// TIA Portal project "ASANSÖR_BANT" (V17)
// Vorlageprojekt für das Buch mit Zielsystem S7-1200

(* hardware
DEVICE "S7-1200-Station_1"  S7-1200 Station
   slot 0: "Baugruppenträger_0"  Rack  V1.0
   slot 1: "PLC_1"  CPU 1214C DC/DC/Rly  6ES7 214-1HG40-0XB0  V4.5
*)

// ===== PLC "PLC_1"  CPU 1214C DC/DC/Rly =====

VAR_GLOBAL   // PLC tag table "Standard-Variablentabelle"
   "START" AT %E0.0 : Bool;
   "STOP" AT %E0.1 : Bool;
   "SENSÖR 1" AT %I0.2 : Bool;
   "SENSÖR 2" AT %I0.3 : Bool;
   "PLAT.LİM.SENSÖR" AT %I0.5 : Bool;
   "ASAN.LİM.SENSÖR" AT %I0.6 : Bool;
   "KONVEYÖR 1" AT %Q0.0 : Bool;
   "KONVEYÖR 2" AT %Q0.1 : Bool;
   "PLAT.İLERİ.HAR." AT %Q0.2 : Bool;
   "PLAT.DÖNDÜR" AT %Q0.3 : Bool;
   "ASAN.İLERİ" AT %Q0.4 : Bool;
   "ASAN.YUKARI" AT %Q0.5 : Bool;
   "SENSÖR 3" AT %I0.4 : Bool;
   "PLAT.DÖNÜŞ.SENSÖR" AT %I0.7 : Bool;
END_VAR

// folder: System blocks/Program resources

DATA_BLOCK "TİMER 1"   // DB1
{ S7_Optimized_Access := 'TRUE' }
AUTHOR : Simatic
FAMILY : IEC
NAME : IEC_TMR
VERSION : 1.0
// stored: InstanceOfName IEC_TIMER
"IEC_TIMER"
BEGIN
END_DATA_BLOCK

// folder: (top level)

FUNCTION "MHJ-PLC-Lab-Function-S71200" : Void   // FC9000, SCL
{ S7_Optimized_Access := 'TRUE' }
VERSION : 0.1
   VAR_TEMP
      rdTimeReturn : Int;
      outputTime : DTL;
      SyncVal : Byte;
      forVal : Int;
      forVal_2 : Int;
      Value : Byte;
   END_VAR
   VAR CONSTANT
      CompVal : Byte := 16#34;
      Value_01 : Byte := 16#11;
      Value_01_DW : DWord := 16#A165_D992;
      Value_02_DW : DWord := 16#58BE_4401;
   END_VAR
BEGIN

   #Value:=PEEK(area := 16#82,
        dbNumber := 0,
        byteOffset := 511);
   #Value := #Value + 1;

   POKE(area := 16#82,
        dbNumber := 0,
        byteOffset := 511,
        value := #Value);

   POKE(area:=16#81,
        dbNumber:=0,
        byteOffset:=1016,
        value:=#Value_01_DW);
   POKE(area := 16#81,
        dbNumber := 0,
        byteOffset := 1020,
        value := #Value_02_DW);

   POKE(area := 16#81,
        dbNumber := 0,
        byteOffset := 511,
        value := B#16#00);

   FOR #forVal := 0 TO 120 DO
       FOR #forVal_2:=0 TO 10 DO
           #rdTimeReturn:=RD_SYS_T(#outputTime);
           #rdTimeReturn := WR_SYS_T(#outputTime);
           #rdTimeReturn := RD_SYS_T(#outputTime);
           #rdTimeReturn := WR_SYS_T(#outputTime);
       END_FOR;
       #SyncVal:= PEEK(area := 16#81,
                      dbNumber := 0,
                      byteOffset := 511);
       IF #SyncVal = #CompVal THEN
          GOTO M_1;
       END_IF;
   END_FOR;
   RETURN;

   M_1:
   POKE(area := 16#81,
        dbNumber := 0,
        byteOffset := 511,
        value := B#16#0);
END_FUNCTION

ORGANIZATION_BLOCK "Main"   // OB1, LAD, ProgramCycle
TITLE = "Main Program Sweep (Cycle)"
{ S7_Optimized_Access := 'TRUE' }
VERSION : 0.1
   VAR_INPUT
      Initial_Call : Bool;   // Initial call of this OB
      Remanence : Bool;   // =True, if remanent data are available
   END_VAR
BEGIN

REGION Network 1: Konnektierungsbaustein für PLC-Lab
   // Im Netzwerk 1 wird der Konnektierungsbaustein für PLC-Lab aufgerufen.
   // Dieser Aufruf darf nicht entfernt werden!
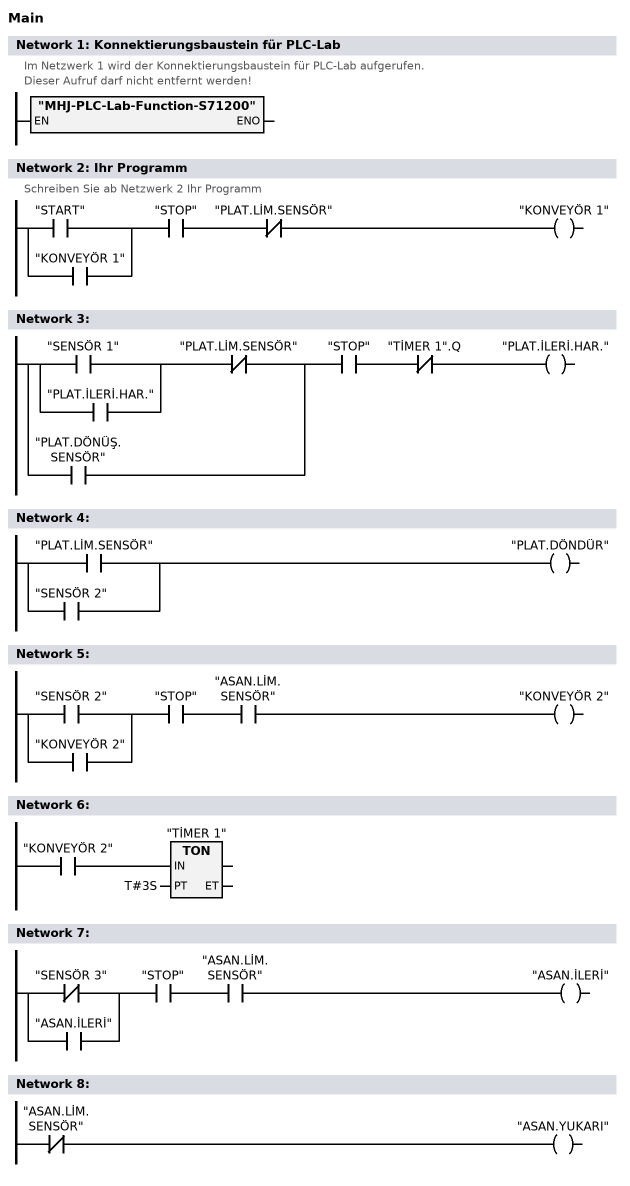
   RUNG wire#powerrail
      "MHJ-PLC-Lab-Function-S71200"()
   END_RUNG
   // the same network as SCL:
   "MHJ-PLC-Lab-Function-S71200"();
END_REGION

REGION Network 2: Ihr Programm
   // Schreiben Sie ab Netzwerk 2 Ihr Programm
   RUNG wire#powerrail
      Contact( "START" )
      wire#w1
      Contact( "STOP" )
      I_Contact( "PLAT.LİM.SENSÖR" )
      Coil( "KONVEYÖR 1" )
   END_RUNG
   RUNG wire#powerrail
      Contact( "KONVEYÖR 1" )
   END_RUNG wire#w1
   // the same network as SCL:
   "KONVEYÖR 1" := ("START" OR "KONVEYÖR 1") AND "STOP" AND NOT "PLAT.LİM.SENSÖR";
END_REGION

REGION Network 3
   RUNG wire#powerrail
      Contact( "SENSÖR 1" )
      wire#w1
      I_Contact( "PLAT.LİM.SENSÖR" )
      wire#w2
      Contact( "STOP" )
      I_Contact( "TİMER 1".Q )
      Coil( "PLAT.İLERİ.HAR." )
   END_RUNG
   RUNG wire#powerrail
      Contact( "PLAT.İLERİ.HAR." )
   END_RUNG wire#w1
   RUNG wire#powerrail
      Contact( "PLAT.DÖNÜŞ.SENSÖR" )
   END_RUNG wire#w2
   // the same network as SCL:
   "PLAT.İLERİ.HAR." := ((("SENSÖR 1" OR "PLAT.İLERİ.HAR.") AND NOT "PLAT.LİM.SENSÖR") OR "PLAT.DÖNÜŞ.SENSÖR") AND "STOP" AND NOT "TİMER 1".Q;
END_REGION

REGION Network 4
   RUNG wire#powerrail
      Contact( "PLAT.LİM.SENSÖR" )
      wire#w1
      Coil( "PLAT.DÖNDÜR" )
   END_RUNG
   RUNG wire#powerrail
      Contact( "SENSÖR 2" )
   END_RUNG wire#w1
   // the same network as SCL:
   "PLAT.DÖNDÜR" := "PLAT.LİM.SENSÖR" OR "SENSÖR 2";
END_REGION

REGION Network 5
   RUNG wire#powerrail
      Contact( "SENSÖR 2" )
      wire#w1
      Contact( "STOP" )
      Contact( "ASAN.LİM.SENSÖR" )
      Coil( "KONVEYÖR 2" )
   END_RUNG
   RUNG wire#powerrail
      Contact( "KONVEYÖR 2" )
   END_RUNG wire#w1
   // the same network as SCL:
   "KONVEYÖR 2" := ("SENSÖR 2" OR "KONVEYÖR 2") AND "STOP" AND "ASAN.LİM.SENSÖR";
END_REGION

REGION Network 6
   "TİMER 1".TON(IN := "KONVEYÖR 2", PT := T#3S);
END_REGION

REGION Network 7
   RUNG wire#powerrail
      I_Contact( "SENSÖR 3" )
      wire#w1
      Contact( "STOP" )
      Contact( "ASAN.LİM.SENSÖR" )
      Coil( "ASAN.İLERİ" )
   END_RUNG
   RUNG wire#powerrail
      Contact( "ASAN.İLERİ" )
   END_RUNG wire#w1
   // the same network as SCL:
   "ASAN.İLERİ" := (NOT "SENSÖR 3" OR "ASAN.İLERİ") AND "STOP" AND "ASAN.LİM.SENSÖR";
END_REGION

REGION Network 8
   RUNG wire#powerrail
      I_Contact( "ASAN.LİM.SENSÖR" )
      Coil( "ASAN.YUKARI" )
   END_RUNG
   // the same network as SCL:
   "ASAN.YUKARI" := NOT "ASAN.LİM.SENSÖR";
END_REGION
END_ORGANIZATION_BLOCK